Universal Robots PolyScope program: Pick_Place_Exam_3.urp

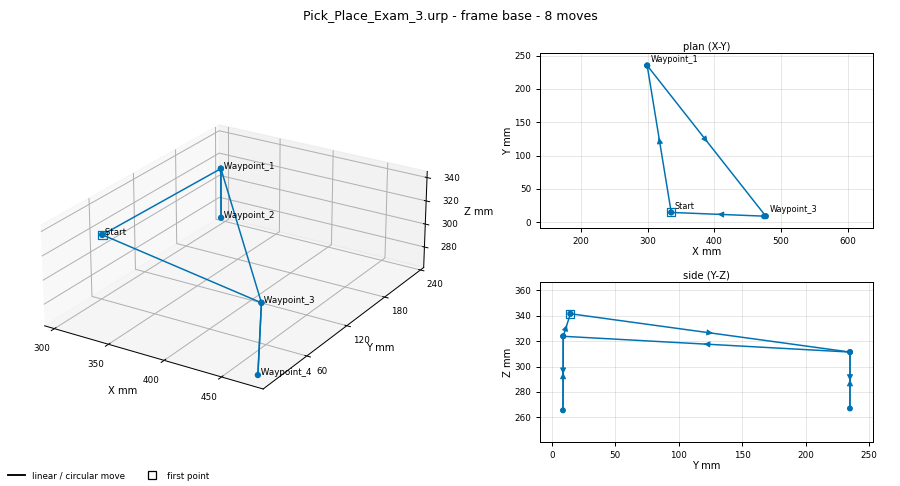
[picture p0: tool path of Pick_Place_Exam_3.urp in frame base, 8 of 8 moves have a stored position in this frame; points joined in program order, loops and branches not executed]
Program Pick_Place_Exam_3 (installation=default directory=/programs/new folder createdIn=5.11.9.1010452 lastSavedIn=5.11.9.1010452 robotSerialNumber=20225200364)
Calibrated DH parameters: a=[0.00002, -0.569483, -0.54992, -0.00001, -0.000036, 0]; d=[0.180894, -146.691669, 192.918669, -46.053088, 0.119778, 0.115602]; alpha=[1.571425, -0.001534, 0.003359, 1.568739, -1.571477, 0]; deltaTheta=[0, 0.376258, -0.101074, -0.275185, -0.000002, 0]
Robot Program (runOnlyOnce=false)
  MoveL speed 250 mm/s, acceleration 1200 mm/s^2 (useActiveTCP=true) feature=Base
    URCap RG Grip (OnRobot, OnRobot A/S) dataModel(rg-target-force=40.0, rg-target-width=0.1, Variable(key=on_return, variable(name=on_return)))
    Waypoint Start: TCP in base x=335.195 y=14.704 z=341.632 mm, rx=-2.1653 ry=2.2518 rz=-0.0236 rad; joints [34.098, -84.1, -131.304, -233.499, -89.502, -143.401] deg
    Waypoint Waypoint_1: TCP in base x=299.172 y=234.982 z=311.443 mm, rx=-2.1898 ry=2.242 rz=0.0149 rad; joints [65.302, -91.603, -128.133, -229.701, -90.522, -113.066] deg
    Waypoint Waypoint_2: TCP in base x=299.228 y=234.909 z=266.998 mm, rx=-2.1893 ry=2.2424 rz=0.0148 rad; joints [65.297, -95.224, -130.249, -223.962, -90.502, -113.029] deg
    URCap RG Grip (OnRobot, OnRobot A/S) dataModel(rg-target-force=40.0, rg-target-width=0.073)
    Waypoint Waypoint_1: TCP in base x=299.172 y=234.982 z=311.443 mm, rx=-2.1898 ry=2.242 rz=0.0149 rad; joints [65.302, -91.603, -128.133, -229.701, -90.522, -113.066] deg
    Waypoint Waypoint_3: TCP in base x=477.035 y=9.023 z=323.881 mm, rx=-2.1897 ry=2.242 rz=0.0149 rad; joints [22.322, -100.119, -116.94, -232.772, -90.829, -156.05] deg
    Waypoint Waypoint_4: TCP in base x=474.395 y=8.828 z=265.501 mm, rx=-2.2179 ry=2.2153 rz=0.0125 rad; joints [22.459, -103.898, -119.739, -226.212, -90.718, -157.312] deg
    URCap RG Grip (OnRobot, OnRobot A/S) dataModel(rg-target-force=40.0, rg-target-width=0.1)
    Waypoint Waypoint_3: TCP in base x=477.035 y=9.023 z=323.881 mm, rx=-2.1897 ry=2.242 rz=0.0149 rad; joints [22.322, -100.119, -116.94, -232.772, -90.829, -156.05] deg
    Waypoint Start: TCP in base x=335.195 y=14.704 z=341.632 mm, rx=-2.1653 ry=2.2518 rz=-0.0236 rad; joints [34.098, -84.1, -131.304, -233.499, -89.502, -143.401] deg
    Halt
